Yaskawa INFORM job: X2_R2_O242(-90,180)NEW.JBI

/JOB
//NAME X2_R2_O242(-90,180)NEW
///FOLDERNAME X4
//POS
///NPOS 129,129,129,4,0,0
///TOOL 0
///POSTYPE PULSE
///PULSE
C00000=-1172,-91659,-106110,-8811,64483,-78082
C00001=-539,-95616,-105965,-5956,62605,-78392
C00002=1085,-105763,-105592,1367,57789,-79187
C00003=48587,-61870,-56373,37554,57186,-71211
C00004=109319,-98863,-81663,-17130,36799,-47258
C00005=110499,-70978,-76585,-14581,28064,-55521
C00006=114923,11399,-23396,-32739,57115,-42289
C00007=112420,58260,23453,-34311,55925,-36712
C00008=103673,61971,28771,-23340,49252,-54180
C00009=104143,61771,30020,-23997,48583,-53787
C00010=104143,61665,31012,-24237,47975,-53623
C00011=104143,61690,30756,-24175,48131,-53665
C00012=104729,63491,32825,-24745,47982,-53345
C00013=104143,61690,30756,-24175,48131,-53665
C00014=107659,59140,34344,-41642,42932,-51759
C00015=107014,61359,36867,-41469,42317,-51817
C00016=107659,59140,34344,-41642,42932,-51759
C00017=114298,50645,22585,-44208,48253,-50722
C00018=115300,57657,31779,-46142,47278,-49521
C00019=115300,57690,33274,-46748,46643,-49118
C00020=115300,57681,32987,-46632,46763,-49196
C00021=114644,58999,34476,-46396,46259,-49299
C00022=115300,57657,31740,-46127,47293,-49533
C00023=110422,53855,26738,-42243,45714,-51626
C00024=110101,51308,25641,-42442,45091,-51468
C00025=110533,52780,27259,-42897,45119,-51216
C00026=110422,53855,26738,-42243,45714,-51626
C00027=116735,58481,29899,-46002,49121,-49762
C00028=118370,75012,51726,-50241,46614,-47038
C00029=118108,70057,46239,-49505,47020,-47507
C00030=118108,70266,48092,-50244,46341,-47020
C00031=118108,70220,47725,-50097,46473,-47117
C00032=117784,71478,49213,-50116,46118,-47086
C00033=118108,70049,46154,-49471,47053,-47531
C00034=118387,83073,57558,-46291,49726,-51230
C00035=118631,86533,63976,-47788,48346,-50211
C00036=118216,85491,62678,-47401,48308,-50455
C00037=118631,86396,63233,-47537,48612,-50383
C00038=116302,66382,28075,-36426,63187,-59231
C00039=111770,60208,27570,-41022,56828,-41847
C00040=97316,77194,43223,-14034,55762,-46071
C00041=111344,65568,37819,-42394,53938,-40685
C00042=111060,67964,39364,-42109,54014,-40875
C00043=96705,67045,31183,-6208,56523,-50696
C00044=96771,67044,31181,-6253,56528,-50671
C00045=98058,64809,28584,-7072,57080,-50206
C00046=102949,69027,31904,-16856,60857,-43628
C00047=110238,88390,54427,-32315,67782,-30590
C00048=111442,81419,52375,-30089,53119,-32051
C00049=110899,64239,29582,-28047,57507,-33617
C00050=117413,74057,37010,-34212,72450,-15391
C00051=110281,62038,31775,-26420,49104,-43606
C00052=106505,97669,59615,-8678,68810,-27055
C00053=106752,100565,64597,-8880,67276,-26852
C00054=109744,62855,32808,-26110,48745,-43759
C00055=107449,68617,39501,-24838,47002,-44382
C00056=109888,61264,27932,-23262,51365,-47452
C00057=117020,70069,39732,-42045,53642,-54528
C00058=116643,71924,44624,-43844,51864,-53336
C00059=118416,82011,56835,-46074,51078,-51852
C00060=118682,82061,56859,-45731,50632,-52022
C00061=119294,90247,68763,-43118,41944,-53035
C00062=119766,73182,44247,-40206,47734,-54839
C00063=120560,63694,30603,-42359,58082,-50105
C00064=116358,64429,23589,-23951,58627,-49139
C00065=116968,-20453,-45092,-25851,41430,-48067
C00066=118489,-78623,-76964,-34127,32976,-43558
C00067=15896,-74508,-72271,73191,84674,-57421
C00068=31461,-74136,-72097,73237,111249,-57325
C00069=37199,-69408,-69826,73614,107600,-56062
C00070=-3643,-76224,-106676,-19950,71810,-76872
C00071=70388,-93367,-87979,22259,92531,-40632
C00072=132234,14944,-6259,12342,59781,-23208
C00073=146205,63473,16177,10072,90044,-15024
C00074=148576,68007,22640,9405,88157,-14412
C00075=148576,67267,23954,9407,86985,-14500
C00076=148576,66783,24956,9411,86132,-14562
C00077=148576,66832,24863,9408,86216,-14555
C00078=149047,69084,27509,9276,85699,-14442
C00079=148423,68574,25700,9447,86607,-14574
C00080=146195,62986,16971,10071,89317,-15086
C00081=176137,58081,9771,-3198,80109,33161
C00082=174052,65626,21441,-2357,76742,32574
C00083=173571,63404,20046,-2157,76447,32425
C00084=173571,63211,20421,-2158,76117,32429
C00085=173571,63292,20263,-2157,76255,32427
C00086=172556,64401,21545,-1729,76012,32099
C00087=173019,62971,18478,-1917,77173,32231
C00088=167045,54371,14180,12829,67421,32117
C00089=167300,57261,17419,12739,66888,32149
C00090=166775,56105,16119,12998,67167,31995
C00091=174959,61653,15361,-2721,78467,32830
C00092=153862,58220,7137,12336,84382,31788
C00093=154888,58914,9595,11964,83110,31986
C00094=146416,53637,12500,29969,73855,35683
C00095=161804,89703,42514,-6671,93266,37768
C00096=160481,83040,34267,-6425,94812,37264
C00097=160461,82996,34213,-6421,94821,37257
C00098=160314,82402,33477,-6393,94958,37204
C00099=155818,71683,20777,1425,95566,24197
C00100=154068,75736,24755,2435,97986,16967
C00101=150406,78568,28210,7412,98870,8330
C00102=143192,78361,31098,15429,92978,3071
C00103=142524,84239,37703,11837,92418,-12035
C00104=142502,84415,37922,11841,92377,-12046
C00105=137937,102743,61702,17663,90401,-30375
C00106=138214,107970,68255,17604,89055,-30475
C00107=138254,108650,69203,17597,88823,-30493
C00108=137728,105908,62856,17713,91318,-30315
C00109=129809,68648,23314,23742,79294,-62187
C00110=130521,38108,-11366,22924,75116,-53839
C00111=144715,56131,10361,11744,72134,27543
C00112=151566,59831,28742,-2859,46138,64220
C00113=152051,66365,37606,-3402,44065,64516
C00114=152470,67516,39026,-3796,43800,64724
C00115=153239,74187,48057,-1867,40213,65616
C00116=151811,68486,39030,4846,43626,66812
C00117=148976,61300,30711,7226,45253,65595
C00118=147729,58500,33654,14300,37151,64277
C00119=144430,59667,36614,25817,36412,63257
C00120=144460,72482,45840,17180,42284,64323
C00121=143111,63918,40413,22730,36091,62179
C00122=143801,66633,41900,20305,38275,63153
C00123=139817,77107,57238,29606,33210,58883
C00124=141383,82478,55565,14874,41935,61497
C00125=144692,57703,21103,13544,52726,73165
C00126=140496,9250,-2578,20724,48099,77689
C00127=103999,-84119,-66645,26288,35960,55555
C00128=-2000,-130321,-133031,0,28968,0
BC00000=196404,515078,981211
BC00001=195624,514960,957134
BC00002=193623,514657,895390
BC00003=148789,507467,173552
BC00004=141590,486355,90511
BC00005=133744,463348,17
BC00006=133744,463348,17
BC00007=133744,463348,17
BC00008=133744,463348,17
BC00009=133744,463348,17
BC00010=133744,463348,17
BC00011=133744,463348,17
BC00012=133744,463348,17
BC00013=133744,463348,17
BC00014=133744,463348,17
BC00015=133744,463348,17
BC00016=133744,463348,17
BC00017=133744,463348,17
BC00018=133744,463348,17
BC00019=133744,463348,17
BC00020=133744,463348,17
BC00021=133744,463348,17
BC00022=133744,463348,17
BC00023=133744,463348,17
BC00024=133744,463348,17
BC00025=133744,463348,17
BC00026=133744,463348,17
BC00027=133744,463348,17
BC00028=133744,463348,17
BC00029=133744,463348,17
BC00030=133744,463348,17
BC00031=133744,463348,17
BC00032=133744,463348,17
BC00033=133744,463348,17
BC00034=133744,463348,17
BC00035=133744,463348,17
BC00036=133744,463348,17
BC00037=133744,463348,17
BC00038=133744,463348,17
BC00039=122188,464291,17
BC00040=122188,464290,17
BC00041=122188,464291,17
BC00042=122188,464291,17
BC00043=122188,464290,17
BC00044=122188,464290,17
BC00045=122188,464290,17
BC00046=122188,464290,17
BC00047=122188,464291,17
BC00048=122188,464291,354
BC00049=122188,464291,354
BC00050=147871,465485,916
BC00051=150420,470888,192
BC00052=151042,472210,17
BC00053=151042,472210,17
BC00054=150420,470888,192
BC00055=150420,470888,192
BC00056=150635,471343,131
BC00057=151043,472209,15
BC00058=151043,472209,15
BC00059=151043,472209,15
BC00060=151042,472209,15
BC00061=151041,472209,15
BC00062=151041,472209,15
BC00063=151043,472209,15
BC00064=150303,469416,10754
BC00065=145083,508024,7369
BC00066=145083,506336,7369
BC00067=139738,502478,3904
BC00068=139738,503304,3904
BC00069=139904,513247,3900
BC00070=199448,515539,1075137
BC00071=258990,522046,241931
BC00072=356760,522046,241931
BC00073=356760,409759,42887
BC00074=356760,409759,42887
BC00075=356760,409759,42887
BC00076=356760,409759,42887
BC00077=356760,409759,42887
BC00078=356760,409759,42887
BC00079=356760,409759,42887
BC00080=356760,409759,42887
BC00081=398158,391605,17411
BC00082=398158,391605,17411
BC00083=398158,391605,17411
BC00084=398158,391605,17411
BC00085=398158,391605,17411
BC00086=398158,391605,17411
BC00087=398158,391605,17411
BC00088=398158,391605,17411
BC00089=398158,391605,17411
BC00090=398158,391605,17411
BC00091=398158,391605,17411
BC00092=344176,409815,17
BC00093=344176,409815,17
BC00094=344176,409815,17
BC00095=344176,409815,17
BC00096=344176,409815,17
BC00097=344176,409815,17
BC00098=344176,409815,17
BC00099=344176,409815,15
BC00100=344176,409815,17
BC00101=344176,409815,17
BC00102=344176,409815,13
BC00103=344176,409815,12
BC00104=344176,409815,12
BC00105=344176,409815,12
BC00106=344176,409815,12
BC00107=344176,409815,12
BC00108=344176,409815,12
BC00109=326504,409815,17
BC00110=326504,409815,17
BC00111=339270,441939,17014
BC00112=344994,456339,24633
BC00113=344994,456339,24633
BC00114=344994,456339,24633
BC00115=344994,456339,24633
BC00116=344994,456339,24631
BC00117=344994,456339,24631
BC00118=344994,456339,24631
BC00119=344994,456339,24631
BC00120=344994,456339,24631
BC00121=344994,456339,24631
BC00122=344994,456339,24631
BC00123=344994,456339,24631
BC00124=344994,456339,24631
BC00125=359830,449275,49809
BC00126=372188,522287,309305
BC00127=335727,515780,471592
BC00128=200118,491577,1075193
EC00000=53467,-715332
EC00001=179590,-335527
EC00002=798141,-184050
EC00003=798073,-185062
EC00004=798113,-184473
EC00005=798156,-183832
EC00006=798156,-183832
EC00007=798156,-183832
EC00008=798156,-183832
EC00009=798156,-183832
EC00010=798156,-183832
EC00011=798156,-183832
EC00012=798156,-183832
EC00013=798156,-183832
EC00014=798156,-183832
EC00015=798156,-183832
EC00016=798156,-183832
EC00017=798156,-183832
EC00018=798156,-183832
EC00019=798156,-183832
EC00020=798156,-183832
EC00021=798156,-183832
EC00022=798156,-183832
EC00023=798156,-183832
EC00024=798156,-183832
EC00025=798156,-183832
EC00026=798156,-183832
EC00027=798156,-183832
EC00028=798156,-183832
EC00029=798156,-183832
EC00030=798156,-183832
EC00031=798156,-183832
EC00032=798156,-183832
EC00033=798156,-183832
EC00034=798156,-183832
EC00035=798156,-183832
EC00036=798156,-183832
EC00037=798156,-183832
EC00038=798156,-183832
EC00039=798156,-183832
EC00040=798153,-183831
EC00041=798156,-183832
EC00042=798156,-183832
EC00043=798153,-183831
EC00044=798153,-183831
EC00045=798153,-183831
EC00046=798154,-183831
EC00047=798156,-183832
EC00048=798156,-183832
EC00049=798156,-183832
EC00050=798156,-183832
EC00051=798155,-183832
EC00052=798156,-183832
EC00053=798156,-183832
EC00054=798155,-183832
EC00055=798155,-183832
EC00056=798155,-183832
EC00057=798155,-183832
EC00058=798155,-183832
EC00059=798155,-183832
EC00060=798150,-183832
EC00061=798153,-183832
EC00062=798153,-183832
EC00063=798155,-183832
EC00064=798155,-183832
EC00065=798155,-183832
EC00066=798155,-183832
EC00067=798155,-183832
EC00068=878588,-403504
EC00069=886883,-1018081
EC00070=798156,-1296783
EC00071=798156,-1296783
EC00072=798156,-1296783
EC00073=798156,-1296783
EC00074=798156,-1296783
EC00075=798156,-1296783
EC00076=798156,-1296783
EC00077=798156,-1296783
EC00078=798156,-1296783
EC00079=798156,-1296783
EC00080=798156,-1296783
EC00081=798156,-1296783
EC00082=798156,-1296783
EC00083=798156,-1296783
EC00084=798156,-1296783
EC00085=798156,-1296783
EC00086=798156,-1296783
EC00087=798156,-1296783
EC00088=798156,-1296783
EC00089=798156,-1296783
EC00090=798156,-1296783
EC00091=798156,-1296783
EC00092=798156,-1296783
EC00093=798156,-1296783
EC00094=798156,-1296783
EC00095=798156,-1296783
EC00096=798156,-1296783
EC00097=798156,-1296783
EC00098=798156,-1296783
EC00099=798155,-1296783
EC00100=798156,-1296783
EC00101=798156,-1296783
EC00102=798154,-1296784
EC00103=798154,-1296784
EC00104=798154,-1296784
EC00105=798154,-1296784
EC00106=798154,-1296784
EC00107=798154,-1296784
EC00108=798154,-1296784
EC00109=798156,-1296783
EC00110=798156,-1296783
EC00111=798156,-1296783
EC00112=798155,-1296783
EC00113=798155,-1296783
EC00114=798155,-1296783
EC00115=798155,-1296783
EC00116=798154,-1296784
EC00117=798154,-1296784
EC00118=798154,-1296784
EC00119=798154,-1296784
EC00120=798154,-1296784
EC00121=798154,-1296784
EC00122=798154,-1296784
EC00123=798154,-1296784
EC00124=798154,-1296784
EC00125=798155,-1296783
EC00126=798155,-1296783
EC00127=798155,-1296783
EC00128=798156,-1296783
///POSTYPE BASE
///RECTAN
///RCONF 0,0,0,0,1,0,0,0,0,0,0,0,0,0,0,0,0,0,0,0,0,0,0,0
P00006=2.006,1.622,-0.565,0.0000,0.0000,0.0000
P00021=0.073,2.058,-0.109,0.0000,0.0000,0.0000
P00022=2.006,1.622,-0.565,0.0000,0.0000,0.0000
///RCONF 0,0,0,0,0,0,0,0,0,0,0,0,0,0,0,0,0,0,0,0,0,0,0,0
P00023=-2.957,-4.083,2.762,0.0000,0.0000,0.0000
//INST
///DATE 2024/12/18 11:57
///ATTR SC,RW
///GROUP1 RB1,BS1
///GROUP2 ST1
NOP
'OK_r2_O24.2(-90,180)
'-90,0
MOVJ C00000 BC00000 VJ=100.00  +MOVJ EC00000 VJ=100.00
MOVJ C00001 BC00001 VJ=100.00  +MOVJ EC00001 VJ=100.00
MOVJ C00002 BC00002 VJ=100.00  +MOVJ EC00002 VJ=100.00
MOVJ C00003 BC00003 VJ=100.00  +MOVJ EC00003 VJ=25.00
MOVJ C00004 BC00004 VJ=100.00  +MOVJ EC00004 VJ=25.00
MOVJ C00005 BC00005 VJ=100.00  +MOVJ EC00005 VJ=100.00
MOVJ C00006 BC00006 VJ=100.00  +MOVJ EC00006 VJ=25.00
'Path S1574
SFTOF3D
MOVJ C00007 BC00007 VJ=100.00  +MOVJ EC00007 VJ=100.00
MOVL C00008 BC00008 V=166.7  +MOVJ EC00008 VJ=100.00
SMOVL C00009 BC00009 V=100.0  +MOVJ EC00009
SREFP 3 C00010 BC00010  +REFP EC00010
CALL JOB:SEARCH-R1-S13D
SET P021 P006
SFTON3D P021
SMOVL C00011 BC00011 V=100.0  +MOVJ EC00011
SREFP 3 C00012 BC00012  +REFP EC00012
CALL JOB:SEARCH-R1-S13D
SET P021 P006
SFTON3D P021
SMOVL C00013 BC00013 V=100.0  +MOVJ EC00013
SMOVL C00014 BC00014 V=200.0  +MOVJ EC00014
SREFP 3 C00015 BC00015  +REFP EC00015
CALL JOB:SEARCH-R1-S13D
SET P021 P006
SFTON3D P021
SMOVL C00016 BC00016 V=100.0  +MOVJ EC00016
SFTOF3D
MOVL C00017 BC00017 V=400.0  +MOVJ EC00017 VJ=100.00
SMOVL C00018 BC00018 V=133.3  +MOVJ EC00018
SREFP 3 C00019 BC00019  +REFP EC00019
CALL JOB:SEARCH-R1-S13D
SET P022 P006
SFTON3D P022
SMOVL C00020 BC00020 V=100.0  +MOVJ EC00020
SREFP 3 C00021 BC00021  +REFP EC00021
CALL JOB:SEARCH-R1-S13D
SET P022 P006
SFTON3D P022
SMOVL C00022 BC00022 V=100.0  +MOVJ EC00022
SMOVL C00023 BC00023 V=200.0  +MOVJ EC00023
SMOVL C00024 BC00024 V=133.3  +MOVJ EC00024
SREFP 3 C00025 BC00025  +REFP EC00025
CALL JOB:SEARCH-R1-S13D
SET P022 P006
SFTON3D P022
SMOVL C00026 BC00026 V=100.0  +MOVJ EC00026
SFTOF3D
SMOVL C00027 BC00027 V=333.3  +MOVJ EC00027
SMOVL C00028 BC00028 V=166.7  +MOVJ EC00028
SMOVL C00029 BC00029 V=100.0  +MOVJ EC00029
SREFP 3 C00030 BC00030  +REFP EC00030
CALL JOB:SEARCH-R1-S13D
SET P023 P006
SFTON3D P023
SMOVL C00031 BC00031 V=100.0  +MOVJ EC00031
SREFP 3 C00032 BC00032  +REFP EC00032
CALL JOB:SEARCH-R1-S13D
SET P023 P006
SFTON3D P023
SMOVL C00033 BC00033 V=100.0  +MOVJ EC00033
SMOVL C00034 BC00034 V=200.0  +MOVJ EC00034
SMOVL C00035 BC00035 V=166.7  +MOVJ EC00035
SREFP 3 C00036 BC00036  +REFP EC00036
CALL JOB:SEARCH-R1-S13D
SET P023 P006
SFTON3D P023
SMOVL C00037 BC00037 V=200.0  +MOVJ EC00037
SFTOF3D
SMOVL C00038 BC00038 V=500.0  +MOVJ EC00038
'Path W1575
SFTOF3D
SFTON3D P021
MOVJ C00039 BC00039 VJ=100.00  +MOVJ EC00039 VJ=100.00
SMOVL C00040 BC00040 V=166.7 PL=0  +MOVJ EC00040
SREFP 1 C00041 BC00041  +REFP EC00041
SREFP 2 C00042 BC00042  +REFP EC00042
MACRO1 MJ#(0) ARGF9
ARCON
SMOVL C00043 BC00043 V=10.0  +MOVJ EC00043
SMOVC C00044 BC00044 V=10.0  +MOVJ EC00044
SMOVC C00045 BC00045 V=10.0  +MOVJ EC00045
SFTON3D P022
SMOVC C00046 BC00046 V=11.0  +MOVJ EC00046
SMOVC C00047 BC00047 V=10.0  +MOVJ EC00047
SFTON3D P023
SMOVL C00048 BC00048 V=10.0  +MOVJ EC00048
ARCOF
SMOVL C00049 BC00049 V=400.0  +MOVJ EC00049
SFTOF3D
'Path W1576
SFTOF3D
SFTON3D P021
SMOVL C00050 BC00050 V=133.3  +MOVJ EC00050
SFTOF3D
SFTON3D P021
SMOVL C00051 BC00051 V=133.3 PL=0  +MOVJ EC00051
SREFP 1 C00052 BC00052  +REFP EC00052
SREFP 2 C00053 BC00053  +REFP EC00053
MACRO1 MJ#(0) ARGF9
ARCON
SMOVL C00054 BC00054 V=7.5  +MOVJ EC00054
SMOVL C00055 BC00055 V=7.5  +MOVJ EC00055
ARCOF
MOVL C00056 BC00056 V=166.7  +MOVJ EC00056 VJ=25.00
SFTOF3D
MOVL C00057 BC00057 V=250.0  +MOVJ EC00057 VJ=25.00
SFTON3D P022
SMOVL C00058 BC00058 V=133.3  +MOVJ EC00058
ARCON
SMOVL C00059 BC00059 V=7.5  +MOVJ EC00059
SMOVL C00060 BC00060 V=7.5  +MOVJ EC00060
ARCON
SFTON3D P023
SMOVL C00061 BC00061 V=7.5  +MOVJ EC00061
ARCOF
SMOVL C00062 BC00062 V=166.7  +MOVJ EC00062
SMOVL C00063 BC00063 V=400.0  +MOVJ EC00063
SFTOF3D
MOVJ C00064 BC00064 VJ=100.00  +MOVJ EC00064 VJ=100.00
MOVJ C00065 BC00065 VJ=100.00  +MOVJ EC00065 VJ=25.00
MOVJ C00066 BC00066 VJ=100.00  +MOVJ EC00066 VJ=25.00
MOVJ C00067 BC00067 VJ=100.00  +MOVJ EC00067 VJ=100.00
'-90,180
MOVJ C00068 BC00068 VJ=100.00  +MOVJ EC00068 VJ=100.00
MOVJ C00069 BC00069 VJ=100.00  +MOVJ EC00069 VJ=100.00
MOVJ C00070 BC00070 VJ=100.00  +MOVJ EC00070 VJ=100.00
CALL JOB:CLEAN-R1_KM_NEW
MOVJ C00071 BC00071 VJ=100.00  +MOVJ EC00071 VJ=100.00
MOVJ C00072 BC00072 VJ=100.00  +MOVJ EC00072 VJ=100.00
'Path S4222
SFTOF3D
MOVJ C00073 BC00073 VJ=100.00  +MOVJ EC00073 VJ=100.00
MOVL C00074 BC00074 V=666.7  +MOVJ EC00074 VJ=100.00
SMOVL C00075 BC00075 V=166.7  +MOVJ EC00075
SREFP 3 C00076 BC00076  +REFP EC00076
CALL JOB:SEARCH-R1-S13D
SET P022 P006
SFTON3D P022
SMOVL C00077 BC00077 V=166.7  +MOVJ EC00077
SREFP 3 C00078 BC00078  +REFP EC00078
CALL JOB:SEARCH-R1-S13D
SET P022 P006
SFTON3D P022
SMOVL C00079 BC00079 V=166.7  +MOVJ EC00079
SFTOF3D
MOVL C00080 BC00080 V=1000.0  +MOVJ EC00080 VJ=100.00
'EndPath S4222
'Path S4223
SFTOF3D
MOVJ C00081 BC00081 VJ=100.00  +MOVJ EC00081 VJ=100.00
MOVL C00082 BC00082 V=666.7  +MOVJ EC00082 VJ=100.00
SMOVL C00083 BC00083 V=166.7  +MOVJ EC00083
SREFP 3 C00084 BC00084  +REFP EC00084
CALL JOB:SEARCH-R1-S13D
SET P021 P006
SFTON3D P021
SMOVL C00085 BC00085 V=166.7  +MOVJ EC00085
SREFP 3 C00086 BC00086  +REFP EC00086
CALL JOB:SEARCH-R1-S13D
SET P021 P006
SFTON3D P021
SMOVL C00087 BC00087 V=166.7  +MOVJ EC00087
SMOVL C00088 BC00088 V=166.7  +MOVJ EC00088
SREFP 3 C00089 BC00089  +REFP EC00089
CALL JOB:SEARCH-R1-S13D
SET P021 P006
SFTON3D P021
SMOVL C00090 BC00090 V=166.7  +MOVJ EC00090
MOVL C00091 BC00091 V=1000.0  +MOVJ EC00091 VJ=100.00
'EndPath S4223
'Path W4224
SFTOF3D
MOVJ C00092 BC00092 VJ=100.00  +MOVJ EC00092 VJ=100.00
SFTON3D P021
MOVL C00093 BC00093 V=666.7  +MOVJ EC00093 VJ=100.00
SMOVL C00094 BC00094 V=166.7 PL=0  +MOVJ EC00094
MACRO1 MJ#(0) ARGF9
ARCON
SMOVL C00095 BC00095 V=10.0  +MOVJ EC00095
SMOVL C00096 BC00096 V=9.2  +MOVJ EC00096
SMOVC C00097 BC00097 V=10.0  +MOVJ EC00097
SMOVC C00098 BC00098 V=10.0  +MOVJ EC00098
SFTON3D P022
SMOVC C00099 BC00099 V=10.0  +MOVJ EC00099
SMOVC C00100 BC00100 V=10.0  +MOVJ EC00100
SMOVC C00101 BC00101 V=10.0  +MOVJ EC00101
SMOVL C00102 BC00102 V=10.0  +MOVJ EC00102
SMOVL C00103 BC00103 V=10.0  +MOVJ EC00103
SMOVC C00104 BC00104 V=9.2  +MOVJ EC00104
SFTON3D P021
SMOVC C00105 BC00105 V=10.0  +MOVJ EC00105
SMOVC C00106 BC00106 V=10.0  +MOVJ EC00106
SMOVL C00107 BC00107 V=10.0  +MOVJ EC00107
ARCOF
MOVL C00108 BC00108 V=800.0  +MOVJ EC00108 VJ=100.00
MOVL C00109 BC00109 V=1000.0  +MOVJ EC00109 VJ=100.00
'EndPath W4224
MOVJ C00110 BC00110 VJ=100.00  +MOVJ EC00110 VJ=100.00
MOVJ C00111 BC00111 VJ=100.00  +MOVJ EC00111 VJ=100.00
'Path W4225
SFTOF3D
SFTON3D P021
SMOVL C00112 BC00112 V=800.0  +MOVJ EC00112
SMOVL C00113 BC00113 V=166.7 PL=0  +MOVJ EC00113
MACRO1 MJ#(0) ARGF21
ARCON
SMOVL C00114 BC00114 V=7.5  +MOVJ EC00114
SMOVL C00115 BC00115 V=7.5  +MOVJ EC00115
ARCOF
SMOVL C00116 BC00116 V=800.0  +MOVJ EC00116
SMOVL C00117 BC00117 V=1000.0  +MOVJ EC00117
SFTOF3D
'EndPath W4225
'Path W4226
SFTOF3D
SFTON3D P022
SMOVL C00118 BC00118 V=166.7 PL=0  +MOVJ EC00118
ARCON
SMOVL C00119 BC00119 V=8.3  +MOVJ EC00119
SMOVL C00120 BC00120 V=8.3  +MOVJ EC00120
ARCOF
SMOVL C00121 BC00121 V=800.0  +MOVJ EC00121
SFTOF3D
'EndPath W4226
'Path W4227
SFTOF3D
SFTON3D P022
SMOVL C00122 BC00122 V=166.7 PL=0  +MOVJ EC00122
ARCON
SMOVL C00123 BC00123 V=7.5  +MOVJ EC00123
ARCOF
SMOVL C00124 BC00124 V=800.0  +MOVJ EC00124
SMOVL C00125 BC00125 V=1000.0  +MOVJ EC00125
SFTOF3D
'EndPath W4227
MOVJ C00126 BC00126 VJ=100.00  +MOVJ EC00126 VJ=100.00
MOVJ C00127 BC00127 VJ=100.00  +MOVJ EC00127 VJ=100.00
MOVJ C00128 BC00128 VJ=100.00  +MOVJ EC00128 VJ=100.00
END
